Staubli VAL3: stop.pgx

program stop()
begin
  popUpMsg("Cycle is end")
  sock="end"
end
